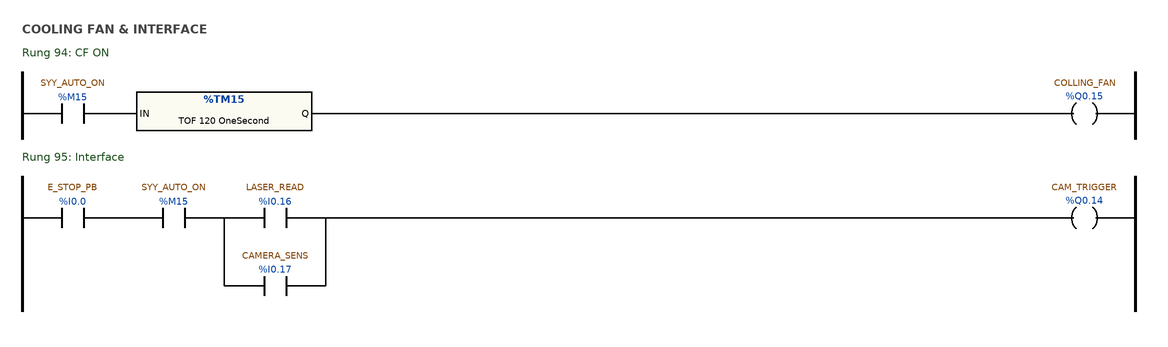
[picture p24: COOLING FAN & INTERFACE, ladder]

// Rung 94: CF ON
  BLK %TM15
  LD %M15                 (* SYY_AUTO_ON *)
  IN
  OUT_BLK
  LD Q
  ST %Q0.15               (* COLLING_FAN *)
  END_BLK
  // as ST:
  //   %TM15(IN := SYY_AUTO_ON);
  //   COLLING_FAN := %TM15.Q;

// Rung 95: Interface
  LD %I0.0                (* E_STOP_PB *)
  AND %M15                (* SYY_AUTO_ON *)
  AND( %I0.16             (* LASER_READ *)
  OR %I0.17               (* CAMERA_SENS *)
  )
  ST %Q0.14               (* CAM_TRIGGER *)
  // as ST:
  //   CAM_TRIGGER := E_STOP_PB AND SYY_AUTO_ON AND (LASER_READ OR CAMERA_SENS);
